Yaskawa INFORM job: profile_program.JBI

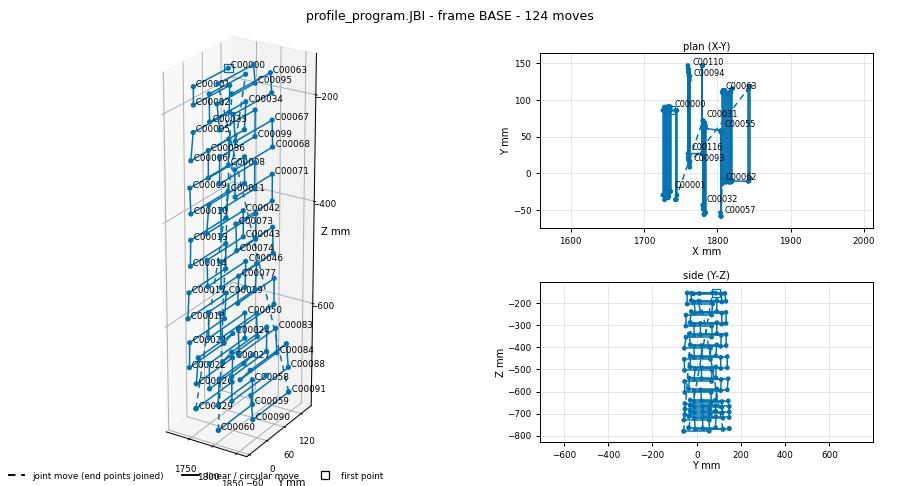
[picture p0: tool path of profile_program.JBI in frame BASE, 124 of 130 moves have a stored position in this frame; points joined in program order, loops and branches not executed]
/JOB
//NAME profile_program
//POS
///NPOS 124,0,124,0,0,0
///TOOL 0
///POSTYPE BASE
///RECTAN
///RCONF 0,0,0,0,0,0,0,0,0,0,0,0,0,0,0,0,0,0,0,0,0,0,0,0
C00000=1736.422403,86.068725,-155.434963,175.000000,-89.999999,5.000000
C00001=1736.422403,-24.535121,-155.434963,175.000000,-89.999999,5.000000
C00002=1736.264297,-24.556340,-188.393261,175.000000,-89.999999,5.000000
C00003=1736.264297,90.766309,-188.393261,175.000000,-89.999999,5.000000
C00004=1735.293262,90.741302,-238.393261,175.000000,-89.999999,5.000000
C00005=1735.293262,-24.591956,-238.393261,175.000000,-89.999999,5.000000
C00006=1734.176386,-30.905387,-288.393261,175.000000,-89.999999,5.000000
C00007=1734.176386,91.064384,-288.393261,175.000000,-89.999999,5.000000
C00008=1733.126465,90.612827,-338.393261,175.000000,-89.999999,5.000000
C00009=1733.126465,-33.383689,-338.393261,175.000000,-89.999999,5.000000
C00010=1732.102746,-29.288229,-388.393261,175.000000,-89.999999,5.000000
C00011=1732.102746,90.993647,-388.393261,175.000000,-89.999999,5.000000
C00012=1731.069150,86.485190,-438.393261,175.000000,-89.999999,5.000000
C00013=1731.069150,-29.104668,-438.393261,175.000000,-89.999999,5.000000
C00014=1730.145389,-29.327342,-488.393261,175.000000,-89.999999,5.000000
C00015=1730.145389,86.362428,-488.393261,175.000000,-89.999999,5.000000
C00016=1729.160231,87.305626,-538.393261,175.000000,-89.999999,5.000000
C00017=1729.160231,-33.308026,-538.393261,175.000000,-89.999999,5.000000
C00018=1728.139861,-35.923342,-588.393261,175.000000,-89.999999,5.000000
C00019=1728.139861,90.590385,-588.393261,175.000000,-89.999999,5.000000
C00020=1727.037759,86.339577,-638.393261,175.000000,-89.999999,5.000000
C00021=1727.037759,-29.255760,-638.393261,175.000000,-89.999999,5.000000
C00022=1725.978021,-29.514401,-688.393261,175.000000,-89.999999,5.000000
C00023=1725.978021,85.894811,-688.393261,175.000000,-89.999999,5.000000
C00024=1745.102078,85.835179,-663.393261,180.000000,-60.000000,0.000000
C00025=1745.102078,-29.657973,-663.393261,180.000000,-60.000000,0.000000
C00026=1744.209099,-35.320140,-713.393261,180.000000,-60.000000,0.000000
C00027=1744.209099,86.263856,-713.393261,180.000000,-60.000000,0.000000
C00028=1743.303053,85.698252,-763.393261,180.000000,-60.000000,0.000000
C00029=1743.303053,-35.923342,-763.393261,180.000000,-60.000000,0.000000
C00030=1743.303053,-35.923342,-763.393261,180.000000,-60.000000,0.000000
C00031=1780.428435,72.066706,-154.024744,175.000000,-89.999999,5.000000
C00032=1780.428435,-43.454005,-154.024744,175.000000,-89.999999,5.000000
C00033=1780.842887,-43.299687,-204.024744,175.000000,-89.999999,5.000000
C00034=1780.842887,72.038891,-204.024744,175.000000,-89.999999,5.000000
C00035=1781.075198,67.207142,-254.024744,175.000000,-89.999999,5.000000
C00036=1781.075198,-48.332654,-254.024744,175.000000,-89.999999,5.000000
C00037=1781.319924,-49.071717,-304.024744,175.000000,-89.999999,5.000000
C00038=1781.319924,67.123641,-304.024744,175.000000,-89.999999,5.000000
C00039=1781.525340,67.123641,-354.024744,175.000000,-89.999999,5.000000
C00040=1781.525340,-48.432624,-354.024744,175.000000,-89.999999,5.000000
C00041=1781.879050,-55.941488,-404.024744,175.000000,-89.999999,5.000000
C00042=1781.879050,62.267743,-404.024744,175.000000,-89.999999,5.000000
C00043=1782.191879,62.005484,-454.024744,175.000000,-89.999999,5.000000
C00044=1782.191879,-56.095428,-454.024744,175.000000,-89.999999,5.000000
C00045=1782.746070,-55.156281,-504.024744,175.000000,-89.999999,5.000000
C00046=1782.746070,69.255697,-504.024744,175.000000,-89.999999,5.000000
C00047=1783.087173,66.963329,-554.024744,175.000000,-89.999999,5.000000
C00048=1783.087173,-54.600457,-554.024744,175.000000,-89.999999,5.000000
C00049=1783.559484,-53.621073,-604.024744,175.000000,-89.999999,5.000000
C00050=1783.559484,65.331526,-604.024744,175.000000,-89.999999,5.000000
C00051=1783.809757,64.991119,-654.024744,175.000000,-89.999999,5.000000
C00052=1783.809757,-53.535884,-654.024744,175.000000,-89.999999,5.000000
C00053=1784.163776,-53.694741,-704.024744,175.000000,-89.999999,5.000000
C00054=1784.163776,61.420216,-704.024744,175.000000,-89.999999,5.000000
C00055=1804.541844,58.271767,-679.024744,180.000000,-60.000000,0.000000
C00056=1804.541844,-53.621539,-679.024744,180.000000,-60.000000,0.000000
C00057=1804.921869,-58.477727,-729.024744,180.000000,-60.000000,0.000000
C00058=1804.921869,57.077374,-729.024744,180.000000,-60.000000,0.000000
C00059=1805.382272,56.614187,-779.024744,180.000000,-60.000000,0.000000
C00060=1805.382272,-58.568269,-779.024744,180.000000,-60.000000,0.000000
C00061=1805.382272,-58.568269,-779.024744,180.000000,-60.000000,0.000000
C00062=1806.741774,-14.564308,-157.833318,175.000000,-89.999999,5.000000
C00063=1806.741774,110.386589,-157.833318,175.000000,-89.999999,5.000000
C00064=1807.935455,113.298523,-195.237262,175.000000,-89.999999,5.000000
C00065=1807.935455,-11.029439,-195.237262,175.000000,-89.999999,5.000000
C00066=1809.223792,-6.975774,-245.237262,175.000000,-89.999999,5.000000
C00067=1809.223792,113.130293,-245.237262,175.000000,-89.999999,5.000000
C00068=1810.433913,113.291353,-295.237262,175.000000,-89.999999,5.000000
C00069=1810.433913,-11.367473,-295.237262,175.000000,-89.999999,5.000000
C00070=1811.720993,-12.074843,-345.237262,175.000000,-89.999999,5.000000
C00071=1811.720993,110.718765,-345.237262,175.000000,-89.999999,5.000000
C00072=1813.018200,108.838448,-395.237262,175.000000,-89.999999,5.000000
C00073=1813.018200,-11.601281,-395.237262,175.000000,-89.999999,5.000000
C00074=1814.339917,-11.264646,-445.237262,175.000000,-89.999999,5.000000
C00075=1814.339917,108.776309,-445.237262,175.000000,-89.999999,5.000000
C00076=1815.693663,108.840314,-495.237262,175.000000,-89.999999,5.000000
C00077=1815.693663,-6.968022,-495.237262,175.000000,-89.999999,5.000000
C00078=1816.894800,-12.141470,-545.237262,175.000000,-89.999999,5.000000
C00079=1816.894800,110.684139,-545.237262,175.000000,-89.999999,5.000000
C00080=1818.151020,108.783829,-595.237262,175.000000,-89.999999,5.000000
C00081=1818.151020,-12.097402,-595.237262,175.000000,-89.999999,5.000000
C00082=1819.413951,-11.542581,-645.237262,175.000000,-89.999999,5.000000
C00083=1819.413951,113.689427,-645.237262,175.000000,-89.999999,5.000000
C00084=1820.711277,115.765166,-695.237262,175.000000,-89.999999,5.000000
C00085=1820.711277,-10.325741,-695.237262,175.000000,-89.999999,5.000000
C00086=1842.094754,-10.775870,-670.237262,180.000000,-60.000000,0.000000
C00087=1842.094754,113.583628,-670.237262,180.000000,-60.000000,0.000000
C00088=1843.385699,118.886251,-720.237262,180.000000,-60.000000,0.000000
C00089=1843.385699,-10.559899,-720.237262,180.000000,-60.000000,0.000000
C00090=1844.821391,-6.276215,-770.237262,180.000000,-60.000000,0.000000
C00091=1844.821391,118.746934,-770.237262,180.000000,-60.000000,0.000000
C00092=1844.821391,118.746934,-770.237262,180.000000,-60.000000,0.000000
C00093=1762.109109,12.459872,-156.484831,175.000000,-89.999999,5.000000
C00094=1762.109109,127.532642,-156.484831,175.000000,-89.999999,5.000000
C00095=1762.657012,132.216532,-191.849847,175.000000,-89.999999,5.000000
C00096=1762.657012,8.358632,-191.849847,175.000000,-89.999999,5.000000
C00097=1762.525253,16.683543,-241.849847,175.000000,-89.999999,5.000000
C00098=1762.525253,132.531278,-241.849847,175.000000,-89.999999,5.000000
C00099=1762.145570,132.906599,-291.849847,175.000000,-89.999999,5.000000
C00100=1762.145570,16.543947,-291.849847,175.000000,-89.999999,5.000000
C00101=1761.833134,17.024416,-341.849847,175.000000,-89.999999,5.000000
C00102=1761.833134,133.077326,-341.849847,175.000000,-89.999999,5.000000
C00103=1761.563628,133.096936,-391.849847,175.000000,-89.999999,5.000000
C00104=1761.563628,21.880314,-391.849847,175.000000,-89.999999,5.000000
C00105=1761.334051,21.863497,-441.849847,175.000000,-89.999999,5.000000
C00106=1761.334051,138.106802,-441.849847,175.000000,-89.999999,5.000000
C00107=1761.155789,138.280090,-491.849847,175.000000,-89.999999,5.000000
C00108=1761.155789,21.687532,-491.849847,175.000000,-89.999999,5.000000
C00109=1760.929028,21.543106,-541.849847,175.000000,-89.999999,5.000000
C00110=1760.929028,142.129720,-541.849847,175.000000,-89.999999,5.000000
C00111=1760.680449,138.116869,-591.849847,175.000000,-89.999999,5.000000
C00112=1760.680449,18.388257,-591.849847,175.000000,-89.999999,5.000000
C00113=1760.348595,21.613516,-641.849847,175.000000,-89.999999,5.000000
C00114=1760.348595,142.780218,-641.849847,175.000000,-89.999999,5.000000
C00115=1760.027843,147.120151,-691.849847,175.000000,-89.999999,5.000000
C00116=1760.027843,27.159189,-691.849847,175.000000,-89.999999,5.000000
C00117=1779.914242,26.953257,-666.849847,180.000000,-60.000000,0.000000
C00118=1779.914242,147.117125,-666.849847,180.000000,-60.000000,0.000000
C00119=1779.788765,147.065802,-716.849847,180.000000,-60.000000,0.000000
C00120=1779.788765,26.786487,-716.849847,180.000000,-60.000000,0.000000
C00121=1779.658663,27.489413,-766.849847,180.000000,-60.000000,0.000000
C00122=1779.658663,146.806016,-766.849847,180.000000,-60.000000,0.000000
C00123=1779.658663,146.806016,-766.849847,180.000000,-60.000000,0.000000
///POSTYPE PULSE
///PULSE
EC00000=0
EC00001=0
EC00002=0
EC00003=0
EC00004=0
EC00005=0
EC00006=0
EC00007=0
EC00008=0
EC00009=0
EC00010=0
EC00011=0
EC00012=0
EC00013=0
EC00014=0
EC00015=0
EC00016=0
EC00017=0
EC00018=0
EC00019=0
EC00020=0
EC00021=0
EC00022=0
EC00023=0
EC00024=0
EC00025=0
EC00026=0
EC00027=0
EC00028=0
EC00029=0
EC00030=92160
EC00031=92160
EC00032=92160
EC00033=92160
EC00034=92160
EC00035=92160
EC00036=92160
EC00037=92160
EC00038=92160
EC00039=92160
EC00040=92160
EC00041=92160
EC00042=92160
EC00043=92160
EC00044=92160
EC00045=92160
EC00046=92160
EC00047=92160
EC00048=92160
EC00049=92160
EC00050=92160
EC00051=92160
EC00052=92160
EC00053=92160
EC00054=92160
EC00055=92160
EC00056=92160
EC00057=92160
EC00058=92160
EC00059=92160
EC00060=92160
EC00061=184320
EC00062=184320
EC00063=184320
EC00064=184320
EC00065=184320
EC00066=184320
EC00067=184320
EC00068=184320
EC00069=184320
EC00070=184320
EC00071=184320
EC00072=184320
EC00073=184320
EC00074=184320
EC00075=184320
EC00076=184320
EC00077=184320
EC00078=184320
EC00079=184320
EC00080=184320
EC00081=184320
EC00082=184320
EC00083=184320
EC00084=184320
EC00085=184320
EC00086=184320
EC00087=184320
EC00088=184320
EC00089=184320
EC00090=184320
EC00091=184320
EC00092=276480
EC00093=276480
EC00094=276480
EC00095=276480
EC00096=276480
EC00097=276480
EC00098=276480
EC00099=276480
EC00100=276480
EC00101=276480
EC00102=276480
EC00103=276480
EC00104=276480
EC00105=276480
EC00106=276480
EC00107=276480
EC00108=276480
EC00109=276480
EC00110=276480
EC00111=276480
EC00112=276480
EC00113=276480
EC00114=276480
EC00115=276480
EC00116=276480
EC00117=276480
EC00118=276480
EC00119=276480
EC00120=276480
EC00121=276480
EC00122=276480
EC00123=368640
//INST
///DATE 2023/01/23 12:19
///ATTR SC,RW,RJ
////FRAME BASE
///GROUP1 RB1,ST1
NOP
MOVJ P009 EX000 VJ=15.00
MOVJ P009 VJ=15.00
MOVJ C00000 EC00000 VJ=15.0
CALL JOB:SPYON
MOVL C00001 EC00001 V=150.0
MOVL C00002 EC00002 V=150.0
MOVL C00003 EC00003 V=150.0
MOVL C00004 EC00004 V=150.0
MOVL C00005 EC00005 V=150.0
MOVL C00006 EC00006 V=150.0
MOVL C00007 EC00007 V=150.0
MOVL C00008 EC00008 V=150.0
MOVL C00009 EC00009 V=150.0
MOVL C00010 EC00010 V=150.0
MOVL C00011 EC00011 V=150.0
MOVL C00012 EC00012 V=150.0
MOVL C00013 EC00013 V=150.0
MOVL C00014 EC00014 V=150.0
MOVL C00015 EC00015 V=150.0
MOVL C00016 EC00016 V=150.0
MOVL C00017 EC00017 V=150.0
MOVL C00018 EC00018 V=150.0
MOVL C00019 EC00019 V=150.0
MOVL C00020 EC00020 V=150.0
MOVL C00021 EC00021 V=150.0
MOVL C00022 EC00022 V=150.0
MOVL C00023 EC00023 V=150.0
MOVL C00024 EC00024 V=150.0
MOVL C00025 EC00025 V=150.0
MOVL C00026 EC00026 V=150.0
MOVL C00027 EC00027 V=150.0
MOVL C00028 EC00028 V=150.0
MOVL C00029 EC00029 V=150.0
CALL JOB:SPYOF
MOVJ P009 VJ=15.00
MOVL C00030 EC00030 V=150.0
MOVJ C00031 EC00031 VJ=15.0
CALL JOB:SPYON
MOVL C00032 EC00032 V=150.0
MOVL C00033 EC00033 V=150.0
MOVL C00034 EC00034 V=150.0
MOVL C00035 EC00035 V=150.0
MOVL C00036 EC00036 V=150.0
MOVL C00037 EC00037 V=150.0
MOVL C00038 EC00038 V=150.0
MOVL C00039 EC00039 V=150.0
MOVL C00040 EC00040 V=150.0
MOVL C00041 EC00041 V=150.0
MOVL C00042 EC00042 V=150.0
MOVL C00043 EC00043 V=150.0
MOVL C00044 EC00044 V=150.0
MOVL C00045 EC00045 V=150.0
MOVL C00046 EC00046 V=150.0
MOVL C00047 EC00047 V=150.0
MOVL C00048 EC00048 V=150.0
MOVL C00049 EC00049 V=150.0
MOVL C00050 EC00050 V=150.0
MOVL C00051 EC00051 V=150.0
MOVL C00052 EC00052 V=150.0
MOVL C00053 EC00053 V=150.0
MOVL C00054 EC00054 V=150.0
MOVL C00055 EC00055 V=150.0
MOVL C00056 EC00056 V=150.0
MOVL C00057 EC00057 V=150.0
MOVL C00058 EC00058 V=150.0
MOVL C00059 EC00059 V=150.0
MOVL C00060 EC00060 V=150.0
CALL JOB:SPYOF
MOVJ P009 VJ=15.00
MOVL C00061 EC00061 V=150.0
MOVJ C00062 EC00062 VJ=15.0
CALL JOB:SPYON
MOVL C00063 EC00063 V=150.0
MOVL C00064 EC00064 V=150.0
MOVL C00065 EC00065 V=150.0
MOVL C00066 EC00066 V=150.0
MOVL C00067 EC00067 V=150.0
MOVL C00068 EC00068 V=150.0
MOVL C00069 EC00069 V=150.0
MOVL C00070 EC00070 V=150.0
MOVL C00071 EC00071 V=150.0
MOVL C00072 EC00072 V=150.0
MOVL C00073 EC00073 V=150.0
MOVL C00074 EC00074 V=150.0
MOVL C00075 EC00075 V=150.0
MOVL C00076 EC00076 V=150.0
MOVL C00077 EC00077 V=150.0
MOVL C00078 EC00078 V=150.0
MOVL C00079 EC00079 V=150.0
MOVL C00080 EC00080 V=150.0
MOVL C00081 EC00081 V=150.0
MOVL C00082 EC00082 V=150.0
MOVL C00083 EC00083 V=150.0
MOVL C00084 EC00084 V=150.0
MOVL C00085 EC00085 V=150.0
MOVL C00086 EC00086 V=150.0
MOVL C00087 EC00087 V=150.0
MOVL C00088 EC00088 V=150.0
MOVL C00089 EC00089 V=150.0
MOVL C00090 EC00090 V=150.0
MOVL C00091 EC00091 V=150.0
CALL JOB:SPYOF
MOVJ P009 VJ=15.00
MOVL C00092 EC00092 V=150.0
MOVJ C00093 EC00093 VJ=15.0
CALL JOB:SPYON
MOVL C00094 EC00094 V=150.0
MOVL C00095 EC00095 V=150.0
MOVL C00096 EC00096 V=150.0
MOVL C00097 EC00097 V=150.0
MOVL C00098 EC00098 V=150.0
MOVL C00099 EC00099 V=150.0
MOVL C00100 EC00100 V=150.0
MOVL C00101 EC00101 V=150.0
MOVL C00102 EC00102 V=150.0
MOVL C00103 EC00103 V=150.0
MOVL C00104 EC00104 V=150.0
MOVL C00105 EC00105 V=150.0
MOVL C00106 EC00106 V=150.0
MOVL C00107 EC00107 V=150.0
MOVL C00108 EC00108 V=150.0
MOVL C00109 EC00109 V=150.0
MOVL C00110 EC00110 V=150.0
MOVL C00111 EC00111 V=150.0
MOVL C00112 EC00112 V=150.0
MOVL C00113 EC00113 V=150.0
MOVL C00114 EC00114 V=150.0
MOVL C00115 EC00115 V=150.0
MOVL C00116 EC00116 V=150.0
MOVL C00117 EC00117 V=150.0
MOVL C00118 EC00118 V=150.0
MOVL C00119 EC00119 V=150.0
MOVL C00120 EC00120 V=150.0
MOVL C00121 EC00121 V=150.0
MOVL C00122 EC00122 V=150.0
CALL JOB:SPYOF
MOVJ P009 VJ=15.00
MOVL C00123 EC00123 V=150.0
END
